Staubli VAL3: onRun.pgx

public program onRun(string& x_sItem[])
  local num i
  local string l_sEvent
  local num l_nId
  local num l_nOffset
  local num l_nMoveId
  local bool l_bToStop
  local InstrItem l_iInstr
  local string l_sPath
  local num l_nResult
  local progItem l_pProgItem
  local num l_nIdEvent
begin
  // save the last item..
  l_nIdEvent=cycleStatus:nEvent
  l_pProgItem=cycleStatus:pCycleProg
  // PROG NAME x_sItem
  call loadCycle(x_sItem,l_nResult)
  // continue
  if l_nResult==0
    // SET THE CALL SUB..
    if isDefined(saveProg:pProg[x_sItem])
      saveProg:pProg[x_sItem].sID="SUB "+x_sItem
      l_nOffset=0
      call cycleStatus:getLastId(l_nMoveId)
      // print to screen define the pCycleProg
      cycleStatus:pCycleProg=saveProg:pProg[x_sItem]
      // execute all the action...
      for i=0 to size(saveProg:pProg[x_sItem].iEvent)-1
        l_iInstr=saveProg:pProg[x_sItem].iEvent[i]
        //
        // INSTRUCTION
        //
        if l_iInstr.sType!=""
          //refresh the cycleStatus
          l_sEvent=l_iInstr.sType+" "+l_iInstr.sData
          ? "ACTION RUNNING,"+l_sEvent+",ID="+toString(".3",getMoveId())+","+toString(".3",clock()-cycleStatus:nTime)+",MoveID="+toString("",l_nMoveId)+",Dist="+toString(".2",l_nOffset)
          call cycleStatus:printLog("  -"+l_sEvent)
          cycleStatus:sToShow=l_sEvent
          cycleStatus:sLastAction=l_sEvent
          cycleStatus:nEvent=i
          //
          // RUN THE ACTION
          //
          call saveData:getPathInstr(l_iInstr.sType,l_sPath)
          instruction:libLoad(l_sPath)
          delay(0)
          call instruction:onRun(l_iInstr.sData)
        else
          l_bToStop=true
        endIf
      endFor
      // reinizialize
      cycleStatus:nEvent=l_nIdEvent
      cycleStatus:pCycleProg=l_pProgItem
      use:bUseRefresh=true
    else
      l_bToStop=true
    endIf
  else
    l_bToStop=true
  endIf
  // check the error...
  if l_bToStop
    // error message
    popUpMsg("SUB not FOUND")
    cycleStatus:bToStop=true
    watch(cycleStatus:bToStop==false,1)
  endIf
end
